Staubli VAL3: _interfacePoint.pgx

program _interfacePoint()
  local string l_sMessage
begin
  //
  // acces to the point interface
  //
  if isKeyPressed(289) and (taskStatus("Point")==-1 or taskStatus("Point")>1)
    if (use:nPage>=100000 and use:nPage<=100009) or (use:nPage>=10000 and use:nPage<=10009)
      // TODO
      l_sMessage="Please exit from the page editor before enter in page POINT...."
      popUpMsg(l_sMessage)
      delay(3)
    else
      // SUSPEND THE TASK INTERFACE
      taskKill("Point")
      taskSuspend("Interface")
      // POINT INTERFACE
      taskCreate "Point",50,point_interface:main()
      bTaskPoint=true
      use:bUseRefresh=true
    endIf
  elseIf (taskStatus("Interface")==0 and taskStatus("Point")==-1) and bTaskPoint
    // TASK RESUME
    bTaskPoint=false
    taskResume("Interface",0)
    use:bUseRefresh=true
  endIf
  // release
  delay(0)
end
